PROGRAM P90_Interlock
VAR_INPUT
	bRecipeRunning : BOOL;
	RecipeStopped : BOOL;
	ManualOperation : BOOL;
	AlarmState : BOOL;
	WarningState : BOOL;
	
	bInductionHeaterMC	: BOOL;
	bThermalBathMC		: BOOL;
	bVacuumPumpMC 		: BOOL;
	bLineHeaterMC 		: BOOL; 
END_VAR
VAR_OUTPUT
	bCoverOperationEnable	: BOOL;
	bDORVacEnable			: BOOL;
	bDORAtmEnable			: BOOL;
	bMaintKey				: BOOL;
	bPowerResetSwitch		: BOOL;
	bMainPowerMonitor		: BOOL;
	bRecipeEnable			: BOOL;
END_VAR	
VAR
	bSafetyGasState			: BOOL;
	bAlarmState				: BOOL;
	bPowerResetLED			: BOOL;
	bUPSMode				: BOOL;

END_VAR

(* Read from Device*)
bMaintKey := GVL_IO.aDigitalInputIO[1].0;
bPowerResetSwitch := GVL_IO.aDigitalInputIO[1].1;
bMainPowerMonitor := GVL_IO.aDigitalInputIO[7].5;



IF ManualOperation THEN
	P92_Maintenance.nCaseSignalTower := 4;
	GVL_IO.aDigitalOutputIO[3].0 := bInductionHeaterMC;
	GVL_IO.aDigitalOutputIO[3].1 := bThermalBathMC;
	GVL_IO.aDigitalOutputIO[3].2 := bVacuumPumpMC;
	GVL_IO.aDigitalOutputIO[3].3 := bLineHeaterMC;
END_IF

// For Test Value
bSafetyGasState := TRUE;

// AND Valve01 = FALSE(H2) AND Valve02 = FALSE(H2) AND Valve03(SiH4) AND Valve04(NH2)
// All MO-Source ByPass Stat
bAlarmState := TRUE;

bCoverOperationEnable := bSafetyGasState AND bAlarmState AND P17_DOROperation.isDOROnState = FALSE; //For Test -P16
// bCoverOpenEnable := ing_Racipe AND bAlarmClear AND isInductionHeater = FAULSE

bDORVacEnable := P16_CoverOperation.isCoverClosed AND bAlarmState AND bSafetyGasState AND P17_DOROperation.isDOROnState = FALSE; //For Test -P17
// add : Vacuum Pump ON
bDORAtmEnable := bAlarmState AND bSafetyGasState AND P17_DOROperation.isDOROnState = TRUE;
// Susceptor Temperature, Vacuum Range > 700Torr

//bRecipeEnable := bMaintKey=FALSE AND bRecipeRunning=FALSE AND P16_CoverOperation.isCoverClosed AND P12_IQ_PLUS.bPumpOn;
bRecipeEnable := TRUE;

(* Out to Device*)
GVL_IO.aDigitalOutputIO[3].7 := bPowerResetLED;
GVL_IO.aDigitalOutputIO[2].4 := bUPSMode;

END_PROGRAM

(* stored: Version 1.1.0.1, ProductVersion 3.1.4026.8
   POU P90_Interlock: Id {c8b81d81-de46-4c7a-a894-4387b2cd9bf7}, SpecialFunc None *)
